(*
	Interlock function for solenoid valve located behind the central turbo pump. 
*)
FUNCTION F_TURBO_PROT_SLND_ILK : BOOL
VAR_INPUT
	ScrollPump : ST_RoughPump;
END_VAR
VAR
END_VAR

F_TURBO_PROT_SLND_ILK := ScrollPump.eState = pumpRUNNING;

END_FUNCTION

(* stored: Version 1.1.0.1, ProductVersion 3.1.4024.2
   POU F_TURBO_PROT_SLND_ILK: Id {2cd3cb76-73f3-4300-a3c4-dd435cd2a0c0}, SpecialFunc None *)
